FUNCTION_BLOCK ConveyorController_HCECC (* HCECC based Conveyor Controller *)
  (* Standard: 61499-2 *)
  (* Version 0.0, 2007-06-26, GDS, University of Auckland *)
  (* Compiler header: package fb.rt.hcecc; #include "PLC_includes.h" *)
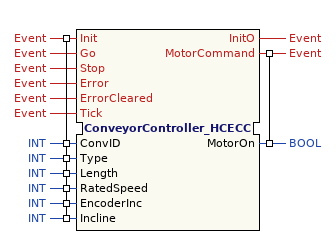
  EVENT_INPUT
    Init WITH ConvID, Type, Length, RatedSpeed, EncoderInc, Incline;
    Go;
    Stop;
    Error;
    ErrorCleared;
    Tick;
  END_EVENT
  EVENT_OUTPUT
    InitO; (* Initialization Confirm *)
    MotorCommand WITH MotorOn;
  END_EVENT
  VAR_INPUT
    ConvID : INT; (* Id of this conveyor *)
    Type : INT;
    Length : INT;
    RatedSpeed : INT;
    EncoderInc : INT;
    Incline : INT; (* CONV_ANGLE_* (-1 DECLINE, 0 LEVEL, 1 INCLINE) *)
  END_VAR
  VAR_OUTPUT
    MotorOn : BOOL; (* true = go, false = stop *)
  END_VAR
  VAR
    ResultCode : INT; (* Return code for a bunch of functions (0 = NoError) *)
    BagsInModel : INT := 0; (* Bags in Model *)
  END_VAR
  ALGORITHM Conv_MotorGo IN C:
void Conv_MotorGo(ConveyorController_HCECC_ECC* me)
{
 me->MotorOn = true;
}
  END_ALGORITHM
  ALGORITHM Conv_MotorStop IN C:
void Conv_MotorStop(ConveyorController_HCECC_ECC* me)
{
 me->MotorOn = false;
}
  END_ALGORITHM
  ALGORITHM InitConveyor IN C:
void InitConveyor(ConveyorController_HCECC_ECC* me)
{
 printf("Conv[%d] InitConv (Empty Function)\n", me->ConvID);
}
  END_ALGORITHM
END_FUNCTION_BLOCK
(* other elements stored in the file *)
(* ECC Name=Conveyor *)
(* ECState Name=START Comment=Initial State *)
(* ECState Name=ERROR Comment=Initialization *)
(* ECAction Algorithm=Conv_LogError *)
(* ECState Name=NORMAL Comment=Normal execution *)
(* ECState Name=INITSTATE *)
(* ECAction Algorithm=InitConveyor *)
(* ECTransition Destination=NORMAL Source=INITSTATE Condition=1 *)
(* ECTransition Destination=ERROR Source=NORMAL Condition=Error *)
(* ECTransition Destination=INITSTATE Source=NORMAL Condition=Init *)
(* ECTransition Destination=ERROR Source=START Condition=Error *)
(* ECTransition Destination=START Source=ERROR Condition=ErrorCleared *)
(* ECTransition Destination=INITSTATE Source=START Condition=Init *)
(* HCECCRelation Destination=BagUpdates Source=Conveyor.NORMAL Relation=Refine Comment=BagRecordECC refines NORMAL of ECC Conveyor *)
(* ECC Name=BagUpdates *)
(* ECState Name=ProcessUpdateQueue *)
(* ECAction Algorithm=Conv_ProcessBagUpdate *)
(* ECTransition Destination=ProcessUpdateQueue Source=ProcessUpdateQueue Condition=1 *)
(* ECC Name=BagExitCheck *)
(* ECState Name=CheckBagExit Comment=Initial State *)
(* ECAction Algorithm=DetectExitBag *)
(* ECTransition Destination=CheckBagExit Source=CheckBagExit Condition=1 *)
(* HCECCRelation Destination=BagExitCheck Source=BagUpdates Relation=Parallel *)
(* ECC Name=BagHandoverCheck *)
(* ECState Name=CheckBagHandover Comment=Initial State *)
(* ECAction Algorithm=HandoverBag *)
(* ECTransition Destination=CheckBagHandover Source=CheckBagHandover Condition=1 *)
(* HCECCRelation Destination=BagHandoverCheck Source=BagUpdates Relation=Parallel *)
